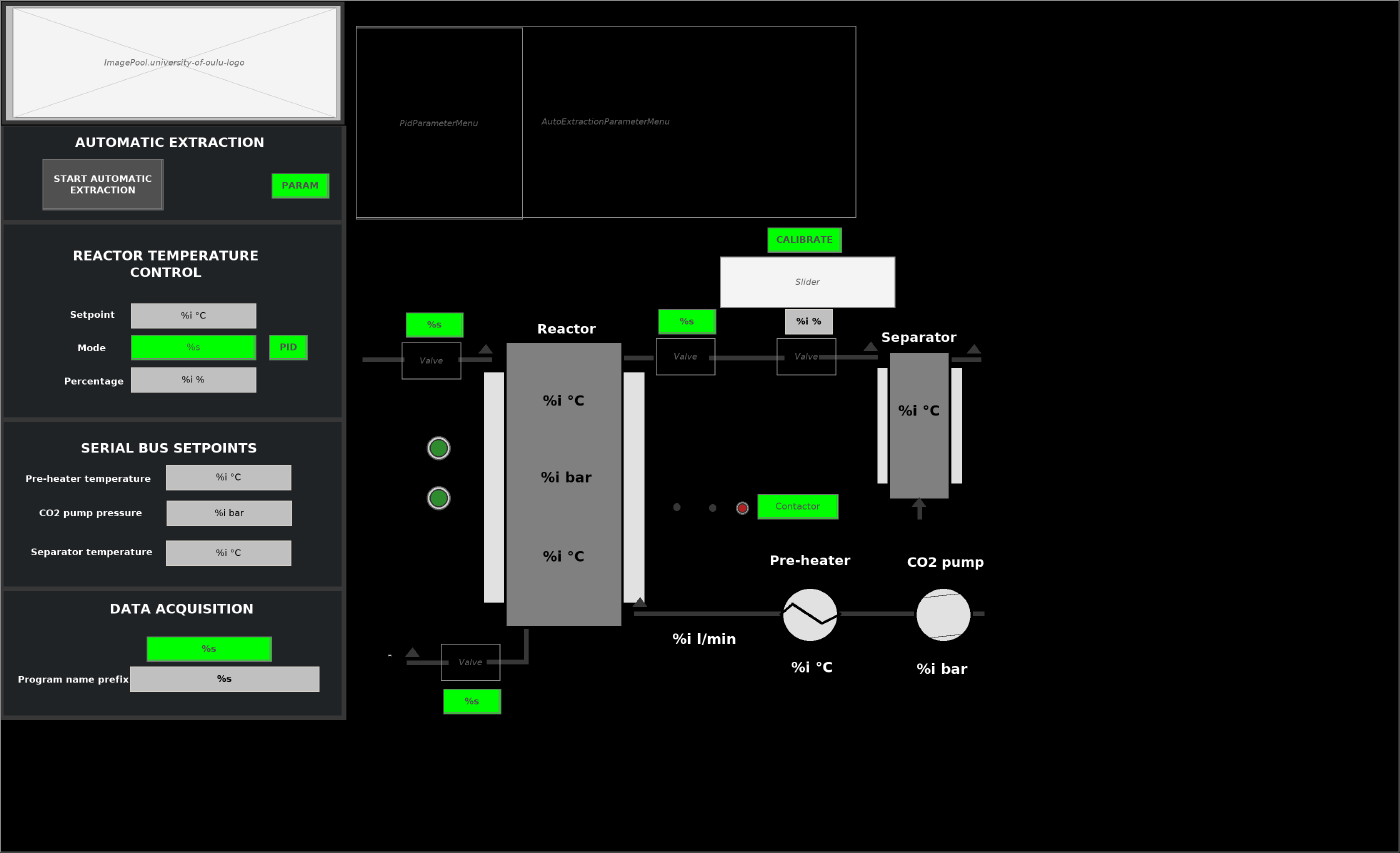
VISUALIZATION MainScreen_1_1  // 1680x1024
    Rectangle (2,151 411x709)
    Textfield (804,746 150x42), "%i l/min", text variable: MainScreenBindings.Co2FlowTextField_TextVariable
    Rectangle (488,793 50x5), colour toggle: MainScreenBindings.SlurryOutLine1_ToggleColor
    Line (604,595) (538,595)
    Line (604,535) (538,535)
    Rectangle (1101,593 5x30)
    Rectangle (831,734 350x5)
    Rectangle (629,755 5x40), colour toggle: MainScreenBindings.SlurryOutLine1_ToggleColor
    Rectangle (584,792 50x5), colour toggle: MainScreenBindings.SlurryOutLine1_ToggleColor
    Rectangle (435,429 50x5), colour toggle: MainScreenBindings.SlurryInArrow_ToggleColor
    Polygon (574,424) (583,413) (591,424) (585,424) (580,424), colour toggle: MainScreenBindings.SlurryInArrow_ToggleColor
    Rectangle (550,429 40x5), colour toggle: MainScreenBindings.SlurryInArrow_ToggleColor
    Rectangle (1050,439 107x144)
    Rectangle (578,444 198x282), colour toggle: MainScreenBindings.ReactorBackgroundRectangle_ToggleColor
    RoundedRectangle (605,409 143x345)
    Button (909,593 97x30), "Contactor", colour toggle: MainScreenBindings.ReactorTemperatureContactorLamp_Variable, invisible if: MainScreenBindings.ReactorTemperatureContactorButton_Invisible
        toggle MainScreenBindings.ReactorTemperatureContactorButton_ToggleVariable p2164770859=TRUE
    Lamp1 (877,601 28x18), variable: MainScreenBindings.ReactorTemperatureContactorLamp_Variable, style: Lamp-Lamp1-Red
    Lamp1 (510,579 33x38), variable: MainScreenBindings.ReactorLowerLevelLamp, style: Lamp-Lamp1-Green
    Lamp1 (510,519 33x38), variable: MainScreenBindings.ReactorUpperLevelLamp_Variable, style: Lamp-Lamp1-Green
    Textfield (157,364 150x30), "%i °C", text variable: MainScreenBindings.ReactorTemperatureSetpointTextField_TextVariable
        OnMouseDown: write the text variable via VisuDialogs.Numpad, min 40, max 120
    Button (157,402 150x30), "%s", text variable: MainScreenBindings.RectorTemperatureControlModeButton_TextVariable, colour toggle: MainScreenBindings.PidParamMenuButton_Invisible
        toggle MainScreenBindings.RectorTemperatureControlModeButton_ToggleVariable
    Label (39,396 142x44), "Mode"
    Label (40,356 142x44), "Setpoint"
    Label (605,380 150x30), "Reactor"
    Image (466,786 3x1), image: VisuSymbols.Symbols.TriangleRight
    Label (42,436 142x44), "Percentage", invisible if: MainScreenBindings.PercentageLabel_Invisible
    Textfield (157,441 150x30), "%i %", text variable: MainScreenBindings.ReactorTemperatureControlPercentageTextField_TextVariable, invisible if: MainScreenBindings.ReactorTemperatureControlPercentageTextField_Invisible
        OnMouseDown: write the text variable via VisuDialogs.Numpad, min 0, max 100
    Label (1975,1166 142x44), "Mode", invisible if: true
    Button (2105,1175 150x30), "%s", text variable: MainScreenBindings.SlurryOutControlModeButton_TextVariable, colour toggle: MainScreenBindings.SlurryOutControlModeButton_ToggleColor, invisible if: true
        toggle MainScreenBindings.SlurryOutControlModeButton_ToggleVariable
    Button (532,827 69x30), "%s", text variable: MainScreenBindings.SlurryOutValveButton_TextVariable, colour toggle: MainScreenBindings.SlurryOutValveButton_ToggleColor, invisible if: MainScreenBindings.SlurryOutValveButton_Invisible
        toggle MainScreenBindings.SlurryOutValveButton_ToggleVariable
    Button (323,402 46x30), "PID", invisible if: MainScreenBindings.PidParamMenuButton_Invisible
        toggle MainScreenBindings.PidParamMenuButton_ToggleVariable
    Frame (427,33 200x230), invisible if: MainScreenBindings.PidParamMenuFrame_Invisible
        shows PidParameterMenu()
    Button (176,764 150x30), "%s", text variable: MainScreenBindings.StartMatlabButton_TextVariable, pressed state: RunMATLAB.bMatlabBtnState, input disabled if: MainScreenBindings.StartMatlabButton_DeactivateInputs
        p2175578022: MainScreenBindings.StartMatlabButton_Color
        toggle MainScreenBindings.StartMatlabButton_ToggleVariable
    Button (487,375 69x30), "%s", text variable: MainScreenBindings.SlurryInValveControlModeButton_TextVariable, colour toggle: MainScreenBindings.SlurryInValveControlModeButton_ToggleColor, invisible if: MainScreenBindings.SlurryInValveControlModeButton_Invisible
        toggle MainScreenBindings.SlurryInValveControlModeButton_ToggleVariable
    Image (2033,1058 2x1), image: VisuSymbols.Symbols.ArrowBoldRight
    Ellipse (937,704 70x68)
    Polyline (936,738) (951,725) (986,748) (1008,737) (1006,737)
    Ellipse (1097,704 70x68)
    Line (1097,718) (1155,712)
    Line (1097,767) (1155,761)
    Textfield (199,558 150x30), "%i °C", text variable: MainScreenBindings.PreHeaterTemperatureSetpointTextField_TextVariable
        OnMouseDown: write MainScreenBindings.PreHeaterTemperatureSetpointTextField_WriteAvariable via VisuDialogs.Numpad, min 0, max 120
    Label (35,553 142x44), "Pre-heater temperature"
    Textfield (200,601 150x30), "%i bar", text variable: MainScreenBindings.Co2PressureSetpointTextField_TextVariable
        OnMouseDown: write MainScreenBindings.Co2PressureSetpointTextField_WriteAvariable via VisuDialogs.Numpad, min 80, max 350
    Label (38,594 142x44), "CO2 pump pressure"
    Label (1060,660 150x30), "CO2 pump"
    Label (906,658 132x30), "Pre-heater"
    RoundedRectangle (1065,421 76x180)
    Label (1028,390 150x30), "Separator"
    Textfield (199,649 150x30), "%i °C", text variable: MainScreenBindings.SeparatorTemperatureSetpointTextField_TextVariable
        OnMouseDown: write MainScreenBindings.SeparatorTemperatureSetpointTextField_WriteAvariable via VisuDialogs.Numpad, min 0, max 100
    Label (39,641 142x44), "Separator temperature"
    Label (2077,957 100x44), "Open time", invisible if: true
    Label (2078,996 100x44), "Closed time", invisible if: true
    Textfield (2174,966 75x30), "%i sec", text variable: MainScreenBindings.SlurryInValveOpenTimeTextField_TextVariable, invisible if: true
        OnMouseDown: write the text variable via VisuDialogs.Numpad, min 0, max 100
    Textfield (2174,1001 75x30), "%i sec", text variable: MainScreenBindings.SlurryInValveClosedTimeTextField_TextVariable, invisible if: true
        OnMouseDown: write the text variable via VisuDialogs.Numpad, min 0, max 200
    Textfield (2139,1048 75x30), "3: %i bar", text variable: MainScreenBindings.UpperIntervalSlurryOffUpperTextField_TextVariable, invisible if: true
        OnMouseDown: write the text variable via VisuDialogs.Numpad, min -100, max 100
    Textfield (2139,1085 75x30), "3: %i bar", text variable: MainScreenBindings.LowerIntervalSlurryOffUpperTextField_TextVariable, invisible if: true
        OnMouseDown: write the text variable via VisuDialogs.Numpad, min -100, max 100
    Label (2141,1116 72x44), "Slurry off + upper", invisible if: true
    Textfield (156,800 227x30), "%s", text variable: MainScreenBindings.ProgramNamePrefixTextField_TextVariable
        OnMouseDown: write the text variable via Edit
    Label (17,794 142x44), "Program name prefix"
    Line (808,609) (775,609)
    Ellipse (807,603 10x11)
    Line (850,609) (817,609), invisible if: MainScreenBindings.ReactorTemperatureContactorClosedLine_Invisible
    Ellipse (850,604 10x11)
    Line (856,594) (823,594), invisible if: MainScreenBindings.ReactorTemperatureContactorOpenLine_Invisible
    Line (877,609) (859,609)
    Frame (482,411 71x44)
        shows Valve(valve_toggleColor := MainScreenBindings.SlurryInValveFrame_valve_toggleColor, valve_tapVariable := MainScreenBindings.SlurryInValveFrame_valve_tapVariable)
    Frame (529,773 71x44)
        shows Valve(valve_toggleColor := MainScreenBindings.SlurryOutValveFrame_valve_toggleColor, valve_tapVariable := MainScreenBindings.SlurryOutValveFrame_valve_tapVariable)
    Polygon (486,788) (495,777) (503,788) (497,788) (492,788), colour toggle: MainScreenBindings.SlurryOutLine1_ToggleColor
    Polygon (759,728) (768,717) (776,728) (770,728) (765,728)
    Rectangle (761,734 75x5)
    Polygon (1036,421) (1045,410) (1053,421) (1047,421) (1042,421), colour toggle: MainScreenBindings.ExtractiveOutLines_ToggleColor
    Rectangle (749,427 35x5), colour toggle: MainScreenBindings.ExtractiveOutLines_ToggleColor
    Polygon (1094,608) (1103,597) (1111,608) (1105,608) (1100,608)
    Rectangle (1142,429 35x5)
    Polygon (1160,424) (1169,413) (1177,424) (1171,424) (1166,424)
    Rectangle (851,427 90x5), colour toggle: MainScreenBindings.ExtractiveOutLines_ToggleColor
    Frame (787,406 71x44)
        shows Valve(valve_toggleColor := MainScreenBindings.ExtractiveOutletOnOff_Valve_ToggleColor, valve_tapVariable := MainScreenBindings.ExtractiveOutletOnOff_Valve_TapVariable)
    Button (790,371 69x30), "%s", text variable: MainScreenBindings.ExtractiveOutOnOffValveButton_TextVariable, colour toggle: MainScreenBindings.ExtractiveOutOnOffValveButton_ToggleColor
        toggle MainScreenBindings.ExtractiveOutOnOffValveButton_ToggleVariable
    Line (985,396) (936,396)
    Rectangle (983,426 70x5), colour toggle: MainScreenBindings.ExtractiveOutLines_ToggleColor
    Frame (932,406 71x44)
        shows Valve(valve_toggleColor := MainScreenBindings.ExtractiveOutletOnOff_Valve_ToggleColor, valve_tapVariable := MainScreenBindings.ExtractiveOutletOnOff_Valve_TapVariable)
    Button (921,273 89x30), "CALIBRATE", invisible if: MainScreenBindings.ExtractiveOutletValveSlider_DisableInputs
        tap MainScreenBindings.ExtractiveOutletValveCalibrateButton_TapVariable
    Slider (864,308 210x61), variable: MainScreenBindings.ExtractiveOutletValveSlider_Variable, invisible if: MainScreenBindings.ExtractiveOutletValveSlider_Invisible, input disabled if: MainScreenBindings.ExtractiveOutletValveSlider_DisableInputs, scale 0..10
    Button (51,191 145x61), "START AUTOMATIC EXTRACTION", text variable: MainScreenBindings.ExtractiveOutOnOffValveButton_TextVariable, colour toggle: MainScreenBindings.StartAutomaticExtractionButton_ToggleVariable, input disabled if: MainScreenBindings.StartAutomaticExtractionButton_DeactivateInputs
        toggle MainScreenBindings.StartAutomaticExtractionButton_ToggleVariable
    Button (326,208 69x30), "PARAM", text variable: MainScreenBindings.SlurryInValveControlModeButton_TextVariable
        toggle MainScreenBindings.autoExtractionParameterMenuButton_ToggleVariable
    Frame (427,31 600x230), invisible if: MainScreenBindings.autoExtractionParameterMenuFrame_Invisible
        shows AutoExtractionParameterMenu()
    Textfield (942,371 57x30), "%i %", text variable: MainScreenBindings.ControlValveOpeningPercentageTextBox_TextVariable
    Rectangle (2,2 411x147)
    Textfield (621,552 117x42), "%i bar", text variable: MainScreenBindings.ReactorPressureTextField_TextVariable
    Textfield (618,647 117x42), "%i °C", text variable: MainScreenBindings.ReactorLowerTemperatureTextField_TextVariable
    Textfield (618,460 117x42), "%i °C", text variable: MainScreenBindings.ReactorUpperTemperatureTextField_TextVariable
    Textfield (916,780 117x42), "%i °C", text variable: MainScreenBindings.PreHeaterTemperatureTextField_TextVariable
    Textfield (1072,782 117x42), "%i bar", text variable: MainScreenBindings.Co2PressureTextField_TextVariable
    Textfield (1072,472 62x42), "%i °C", text variable: MainScreenBindings.SeperatorTemperatureTextField_TextVariable
    Image (15,9 389x132), image: ImagePool.university-of-oulu-logo
    Label (49,156 310x30), "AUTOMATIC EXTRACTION"
    Rectangle (410,151 5x713)
    Label (44,276 310x82), "REACTOR TEMPERATURE CONTROL"
    Label (2,497 402x82), "SERIAL BUS SETPOINTS"
    Label (63,690 310x82), "DATA ACQUISITION"
    Rectangle (-1,264 410x5)
    Rectangle (4,501 410x5)
    Rectangle (1,704 410x5)
    Rectangle (4,859 410x5)
    Rectangle (-1,151 5x713)
END_VISUALIZATION

(* stored: Version 1.1.0.1, ProductVersion 3.1.4024.9
   Visu MainScreen_1_1: Id {3e9d1ae6-676d-4aed-86fb-940379dd364b} *)
